// TIA Portal V17 export
// export: Created 2022-01-19T03:00:58.0499847Z, ExportSetting WithDefaults, DisplayName Totally Integrated Automation Portal, DisplayVersion V17, DisplayName TIA Portal Openness, DisplayVersion V17, DisplayName TIA Portal Teamcenter Gateway, DisplayVersion V17, DisplayName TIA Portal Version Control Interface, DisplayVersion V17, DisplayName TIA Portal Test Suite Advanced, DisplayVersion V17, DisplayName SINAMICS Startdrive Advanced, DisplayVersion V17, DisplayName SINAMICS Startdrive G130, G150, S120, S150, SINAMICS MV, S210, DisplayVersion V17, DisplayName SINAMICS Startdrive G110M, G120, G120C, G120D, G120P, G115D, DisplayVersion V17, DisplayName STEP 7 Professional, DisplayVersion V17, DisplayName STEP 7 Safety, DisplayVersion V17, DisplayName WinCC Professional, DisplayVersion V17, DisplayName SIMATIC Visualization Architect, DisplayVersion V17
FUNCTION_BLOCK "Block_1"   // FB3, LAD
{ S7_Optimized_Access := 'TRUE' }
VERSION : 0.1
// stored: AutoNumber true, IsIECCheckEnabled false, IsRetainMemResEnabled false, MemoryReserve 100, SetENOAutomatically false, UDAEnableTagReadback false
   VAR_INPUT
      "a" : Bool;
   END_VAR
   VAR_OUTPUT
      "b" : Bool;
   END_VAR
   VAR_IN_OUT
      c : Bool;
   END_VAR
   VAR
      d : Bool;
   END_VAR
   VAR_TEMP
      "e" : Bool;
   END_VAR
   VAR CONSTANT
      f : Bool;
   END_VAR
BEGIN

REGION Network 1
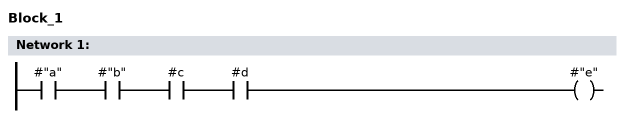
   RUNG wire#powerrail
      Contact( #"a" )
      Contact( #"b" )
      Contact( #c )
      Contact( #d )
      Coil( #"e" )
   END_RUNG
   // the same network as SCL:
   #"e" := #"a" AND #"b" AND #c AND #d;
END_REGION
END_FUNCTION_BLOCK
